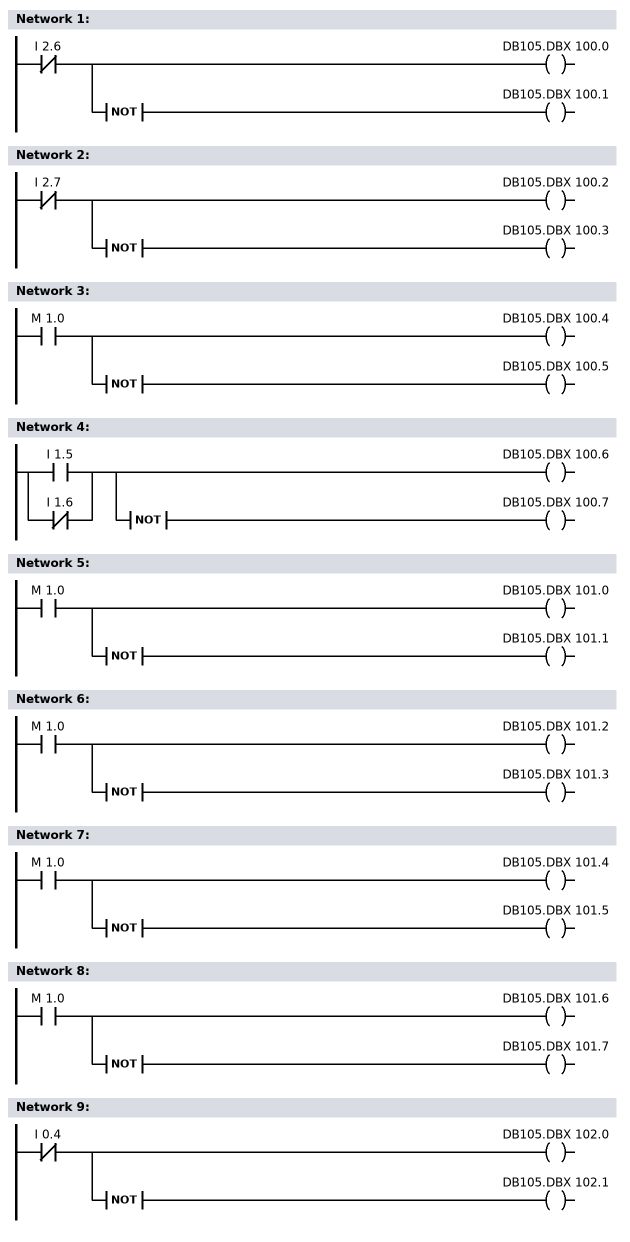
NETWORK
TITLE =
      AN    I 2.6;
      =     L 22.0;
      A     L 22.0;
      BLD   102;
      =     DB105.DBX 100.0;
      A     L 22.0;
      NOT;
      =     DB105.DBX 100.1;
NETWORK
TITLE =
      AN    I 2.7;
      =     L 22.0;
      A     L 22.0;
      BLD   102;
      =     DB105.DBX 100.2;
      A     L 22.0;
      NOT;
      =     DB105.DBX 100.3;
NETWORK
TITLE =
      A     M 1.0;
      =     L 22.0;
      A     L 22.0;
      BLD   102;
      =     DB105.DBX 100.4;
      A     L 22.0;
      NOT;
      =     DB105.DBX 100.5;
NETWORK
TITLE =
      O     I 1.5;
      ON    I 1.6;
      =     L 22.0;
      A     L 22.0;
      BLD   102;
      =     DB105.DBX 100.6;
      A     L 22.0;
      NOT;
      =     DB105.DBX 100.7;
NETWORK
TITLE =
      A     M 1.0;
      =     L 22.0;
      A     L 22.0;
      BLD   102;
      =     DB105.DBX 101.0;
      A     L 22.0;
      NOT;
      =     DB105.DBX 101.1;
NETWORK
TITLE =
      A     M 1.0;
      =     L 22.0;
      A     L 22.0;
      BLD   102;
      =     DB105.DBX 101.2;
      A     L 22.0;
      NOT;
      =     DB105.DBX 101.3;
NETWORK
TITLE =
      A     M 1.0;
      =     L 22.0;
      A     L 22.0;
      BLD   102;
      =     DB105.DBX 101.4;
      A     L 22.0;
      NOT;
      =     DB105.DBX 101.5;
NETWORK
TITLE =
      A     M 1.0;
      =     L 22.0;
      A     L 22.0;
      BLD   102;
      =     DB105.DBX 101.6;
      A     L 22.0;
      NOT;
      =     DB105.DBX 101.7;
NETWORK
TITLE =
      AN    I 0.4;
      =     L 22.0;
      A     L 22.0;
      BLD   102;
      =     DB105.DBX 102.0;
      A     L 22.0;
      NOT;
      =     DB105.DBX 102.1;
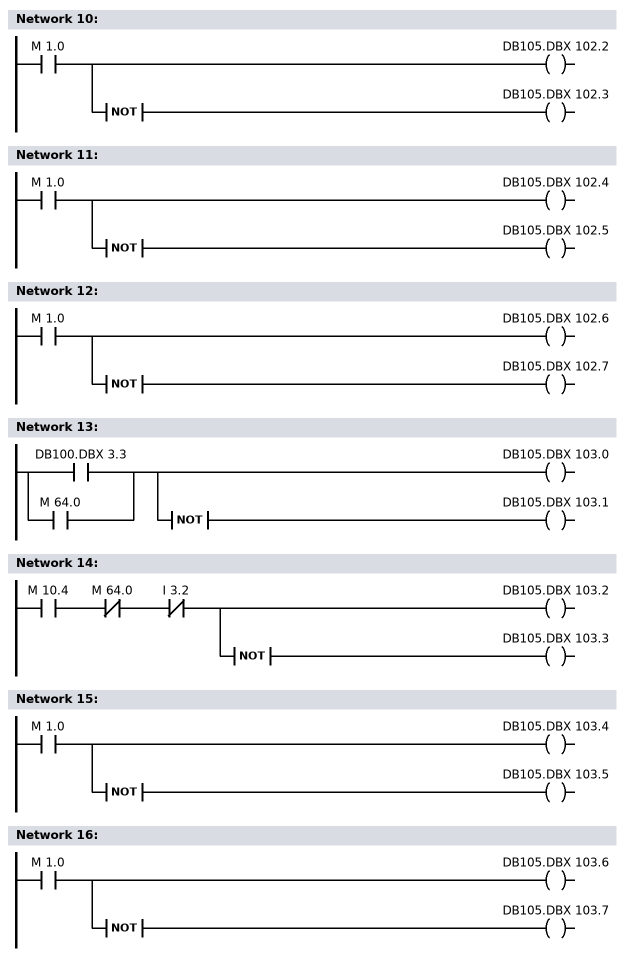
NETWORK
TITLE =
      A     M 1.0;
      =     L 22.0;
      A     L 22.0;
      BLD   102;
      =     DB105.DBX 102.2;
      A     L 22.0;
      NOT;
      =     DB105.DBX 102.3;
NETWORK
TITLE =
      A     M 1.0;
      =     L 22.0;
      A     L 22.0;
      BLD   102;
      =     DB105.DBX 102.4;
      A     L 22.0;
      NOT;
      =     DB105.DBX 102.5;
NETWORK
TITLE =
      A     M 1.0;
      =     L 22.0;
      A     L 22.0;
      BLD   102;
      =     DB105.DBX 102.6;
      A     L 22.0;
      NOT;
      =     DB105.DBX 102.7;
NETWORK
TITLE =
      O     DB100.DBX 3.3;
      O     M 64.0;
      =     L 22.0;
      A     L 22.0;
      BLD   102;
      =     DB105.DBX 103.0;
      A     L 22.0;
      NOT;
      =     DB105.DBX 103.1;
NETWORK
TITLE =
      A     M 10.4;
      AN    M 64.0;
      AN    I 3.2;
      =     L 22.0;
      A     L 22.0;
      BLD   102;
      =     DB105.DBX 103.2;
      A     L 22.0;
      NOT;
      =     DB105.DBX 103.3;
NETWORK
TITLE =
      A     M 1.0;
      =     L 22.0;
      A     L 22.0;
      BLD   102;
      =     DB105.DBX 103.4;
      A     L 22.0;
      NOT;
      =     DB105.DBX 103.5;
NETWORK
TITLE =
      A     M 1.0;
      =     L 22.0;
      A     L 22.0;
      BLD   102;
      =     DB105.DBX 103.6;
      A     L 22.0;
      NOT;
      =     DB105.DBX 103.7;
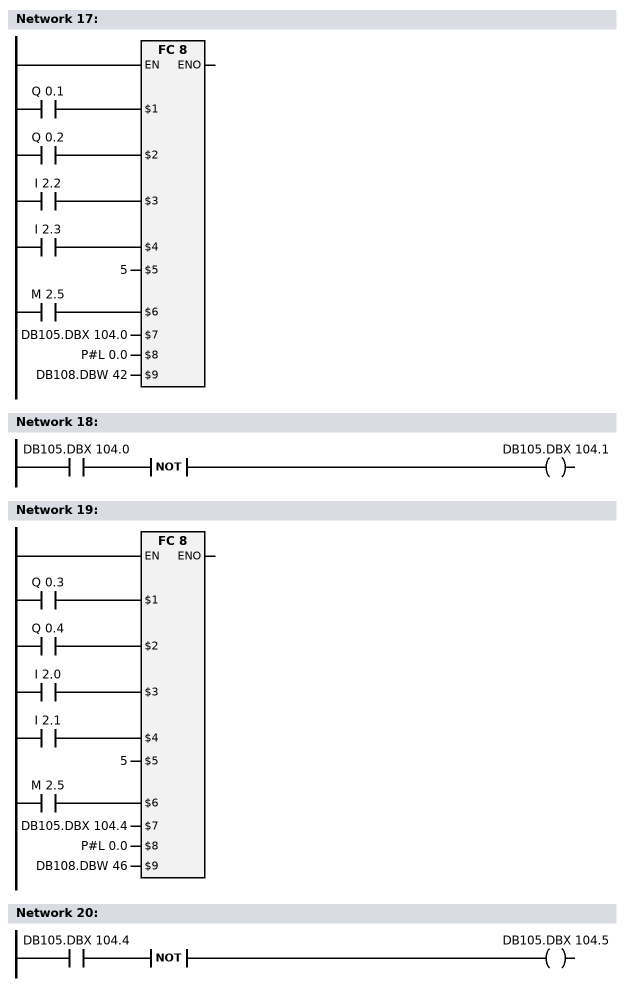
NETWORK
TITLE =
      A     Q 0.1;
      =     L 22.0;
      BLD   103;
      A     Q 0.2;
      =     L 22.1;
      BLD   103;
      A     I 2.2;
      =     L 22.2;
      BLD   103;
      A     I 2.3;
      =     L 22.3;
      BLD   103;
      A     M 2.5;
      =     L 22.4;
      BLD   103;
      CALL  FC 8 (
           $1                       := L 22.0,
           $2                       := L 22.1,
           $3                       := L 22.2,
           $4                       := L 22.3,
           $5                       := 5,
           $6                       := L 22.4,
           $7                       := DB105.DBX 104.0,
           $8                       := P#L 0.0,
           $9                       := DB108.DBW 42);
      NOP   0;
NETWORK
TITLE =
      A     DB105.DBX 104.0;
      NOT;
      =     DB105.DBX 104.1;
NETWORK
TITLE =
      A     Q 0.3;
      =     L 22.0;
      BLD   103;
      A     Q 0.4;
      =     L 22.1;
      BLD   103;
      A     I 2.0;
      =     L 22.2;
      BLD   103;
      A     I 2.1;
      =     L 22.3;
      BLD   103;
      A     M 2.5;
      =     L 22.4;
      BLD   103;
      CALL  FC 8 (
           $1                       := L 22.0,
           $2                       := L 22.1,
           $3                       := L 22.2,
           $4                       := L 22.3,
           $5                       := 5,
           $6                       := L 22.4,
           $7                       := DB105.DBX 104.4,
           $8                       := P#L 0.0,
           $9                       := DB108.DBW 46);
      NOP   0;
NETWORK
TITLE =
      A     DB105.DBX 104.4;
      NOT;
      =     DB105.DBX 104.5;
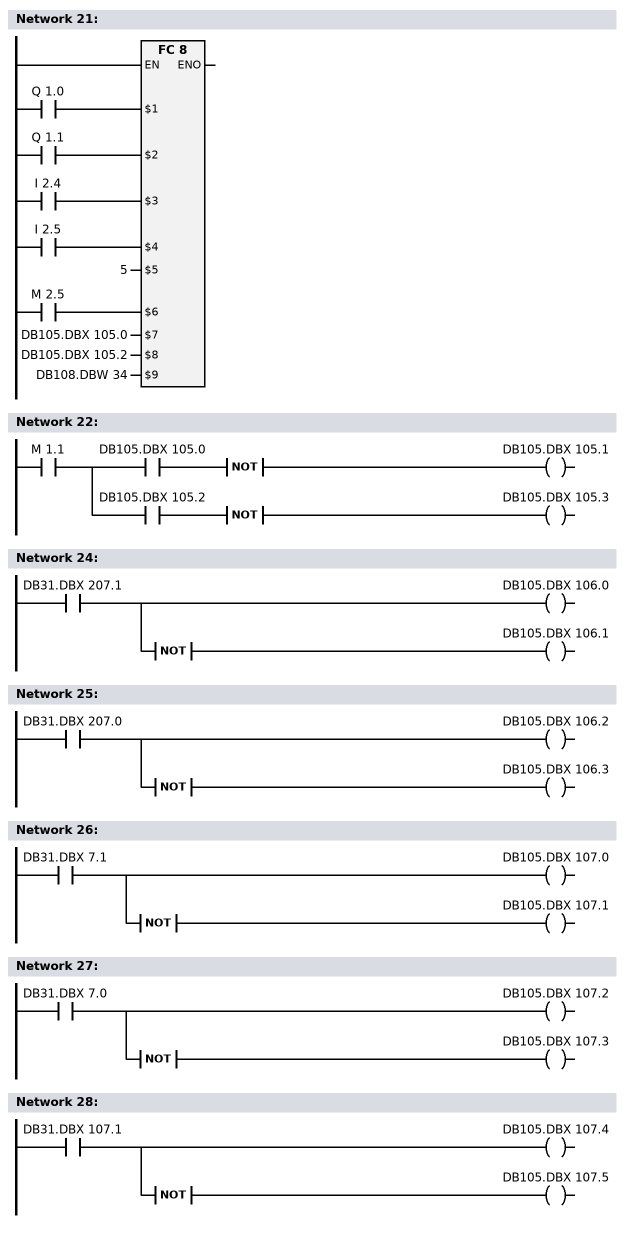
NETWORK
TITLE =
      A     Q 1.0;
      =     L 22.0;
      BLD   103;
      A     Q 1.1;
      =     L 22.1;
      BLD   103;
      A     I 2.4;
      =     L 22.2;
      BLD   103;
      A     I 2.5;
      =     L 22.3;
      BLD   103;
      A     M 2.5;
      =     L 22.4;
      BLD   103;
      CALL  FC 8 (
           $1                       := L 22.0,
           $2                       := L 22.1,
           $3                       := L 22.2,
           $4                       := L 22.3,
           $5                       := 5,
           $6                       := L 22.4,
           $7                       := DB105.DBX 105.0,
           $8                       := DB105.DBX 105.2,
           $9                       := DB108.DBW 34);
      NOP   0;
NETWORK
TITLE =
      A     M 1.1;
      =     L 22.0;
      A     L 22.0;
      A     DB105.DBX 105.0;
      NOT;
      =     DB105.DBX 105.1;
      A     L 22.0;
      A     DB105.DBX 105.2;
      NOT;
      =     DB105.DBX 105.3;
NETWORK
TITLE =
NETWORK
TITLE =
      A     DB31.DBX 207.1;
      =     L 22.0;
      A     L 22.0;
      BLD   102;
      =     DB105.DBX 106.0;
      A     L 22.0;
      NOT;
      =     DB105.DBX 106.1;
NETWORK
TITLE =
      A     DB31.DBX 207.0;
      =     L 22.0;
      A     L 22.0;
      BLD   102;
      =     DB105.DBX 106.2;
      A     L 22.0;
      NOT;
      =     DB105.DBX 106.3;
NETWORK
TITLE =
      A     DB31.DBX 7.1;
      =     L 22.0;
      A     L 22.0;
      BLD   102;
      =     DB105.DBX 107.0;
      A     L 22.0;
      NOT;
      =     DB105.DBX 107.1;
NETWORK
TITLE =
      A     DB31.DBX 7.0;
      =     L 22.0;
      A     L 22.0;
      BLD   102;
      =     DB105.DBX 107.2;
      A     L 22.0;
      NOT;
      =     DB105.DBX 107.3;
NETWORK
TITLE =
      A     DB31.DBX 107.1;
      =     L 22.0;
      A     L 22.0;
      BLD   102;
      =     DB105.DBX 107.4;
      A     L 22.0;
      NOT;
      =     DB105.DBX 107.5;
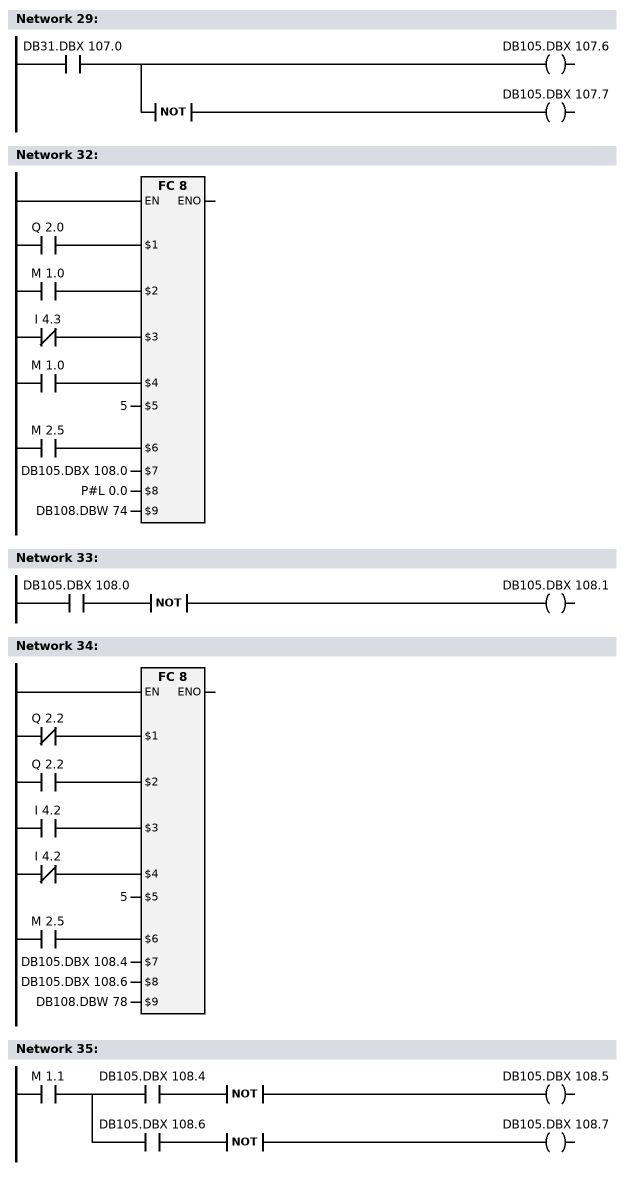
NETWORK
TITLE =
      A     DB31.DBX 107.0;
      =     L 22.0;
      A     L 22.0;
      BLD   102;
      =     DB105.DBX 107.6;
      A     L 22.0;
      NOT;
      =     DB105.DBX 107.7;
NETWORK
TITLE =
NETWORK
TITLE =
NETWORK
TITLE =
      A     Q 2.0;
      =     L 22.0;
      BLD   103;
      A     M 1.0;
      =     L 22.1;
      BLD   103;
      AN    I 4.3;
      =     L 22.2;
      BLD   103;
      A     M 1.0;
      =     L 22.3;
      BLD   103;
      A     M 2.5;
      =     L 22.4;
      BLD   103;
      CALL  FC 8 (
           $1                       := L 22.0,
           $2                       := L 22.1,
           $3                       := L 22.2,
           $4                       := L 22.3,
           $5                       := 5,
           $6                       := L 22.4,
           $7                       := DB105.DBX 108.0,
           $8                       := P#L 0.0,
           $9                       := DB108.DBW 74);
      NOP   0;
NETWORK
TITLE =
      A     DB105.DBX 108.0;
      NOT;
      =     DB105.DBX 108.1;
NETWORK
TITLE =
      AN    Q 2.2;
      =     L 22.0;
      BLD   103;
      A     Q 2.2;
      =     L 22.1;
      BLD   103;
      A     I 4.2;
      =     L 22.2;
      BLD   103;
      AN    I 4.2;
      =     L 22.3;
      BLD   103;
      A     M 2.5;
      =     L 22.4;
      BLD   103;
      CALL  FC 8 (
           $1                       := L 22.0,
           $2                       := L 22.1,
           $3                       := L 22.2,
           $4                       := L 22.3,
           $5                       := 5,
           $6                       := L 22.4,
           $7                       := DB105.DBX 108.4,
           $8                       := DB105.DBX 108.6,
           $9                       := DB108.DBW 78);
      NOP   0;
NETWORK
TITLE =
      A     M 1.1;
      =     L 22.0;
      A     L 22.0;
      A     DB105.DBX 108.4;
      NOT;
      =     DB105.DBX 108.5;
      A     L 22.0;
      A     DB105.DBX 108.6;
      NOT;
      =     DB105.DBX 108.7;
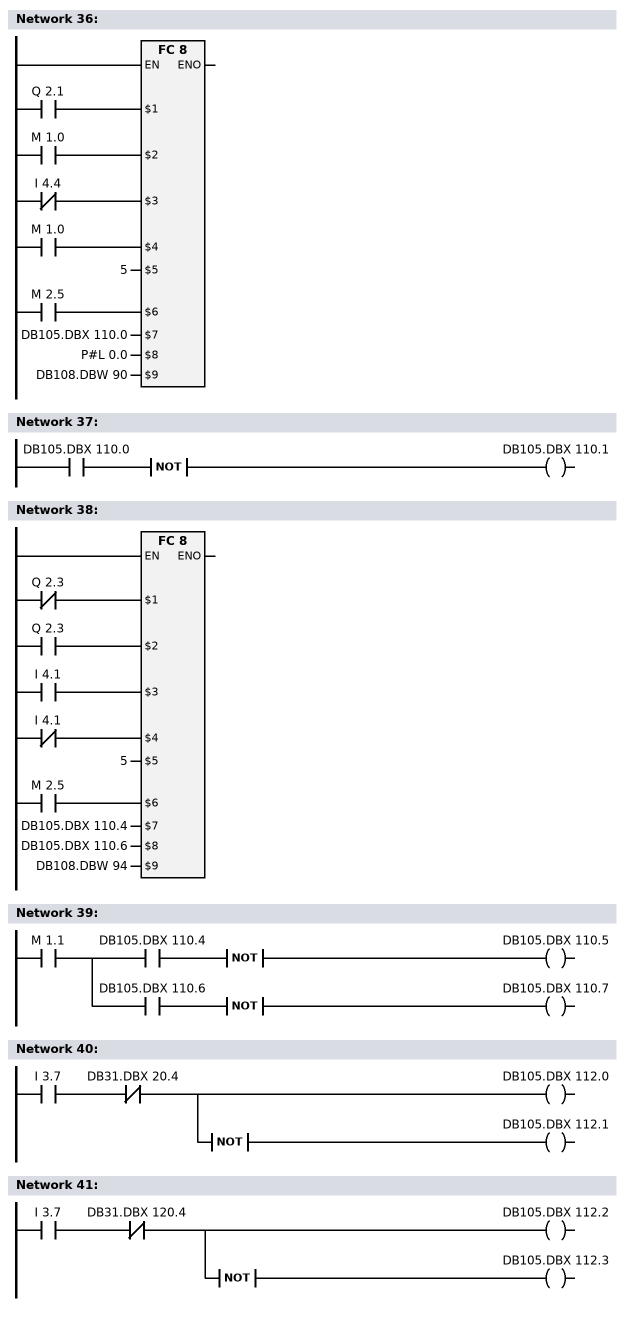
NETWORK
TITLE =
      A     Q 2.1;
      =     L 22.0;
      BLD   103;
      A     M 1.0;
      =     L 22.1;
      BLD   103;
      AN    I 4.4;
      =     L 22.2;
      BLD   103;
      A     M 1.0;
      =     L 22.3;
      BLD   103;
      A     M 2.5;
      =     L 22.4;
      BLD   103;
      CALL  FC 8 (
           $1                       := L 22.0,
           $2                       := L 22.1,
           $3                       := L 22.2,
           $4                       := L 22.3,
           $5                       := 5,
           $6                       := L 22.4,
           $7                       := DB105.DBX 110.0,
           $8                       := P#L 0.0,
           $9                       := DB108.DBW 90);
      NOP   0;
NETWORK
TITLE =
      A     DB105.DBX 110.0;
      NOT;
      =     DB105.DBX 110.1;
NETWORK
TITLE =
      AN    Q 2.3;
      =     L 22.0;
      BLD   103;
      A     Q 2.3;
      =     L 22.1;
      BLD   103;
      A     I 4.1;
      =     L 22.2;
      BLD   103;
      AN    I 4.1;
      =     L 22.3;
      BLD   103;
      A     M 2.5;
      =     L 22.4;
      BLD   103;
      CALL  FC 8 (
           $1                       := L 22.0,
           $2                       := L 22.1,
           $3                       := L 22.2,
           $4                       := L 22.3,
           $5                       := 5,
           $6                       := L 22.4,
           $7                       := DB105.DBX 110.4,
           $8                       := DB105.DBX 110.6,
           $9                       := DB108.DBW 94);
      NOP   0;
NETWORK
TITLE =
      A     M 1.1;
      =     L 22.0;
      A     L 22.0;
      A     DB105.DBX 110.4;
      NOT;
      =     DB105.DBX 110.5;
      A     L 22.0;
      A     DB105.DBX 110.6;
      NOT;
      =     DB105.DBX 110.7;
NETWORK
TITLE =
      A     I 3.7;
      AN    DB31.DBX 20.4;
      =     L 22.0;
      A     L 22.0;
      BLD   102;
      =     DB105.DBX 112.0;
      A     L 22.0;
      NOT;
      =     DB105.DBX 112.1;
NETWORK
TITLE =
      A     I 3.7;
      AN    DB31.DBX 120.4;
      =     L 22.0;
      A     L 22.0;
      BLD   102;
      =     DB105.DBX 112.2;
      A     L 22.0;
      NOT;
      =     DB105.DBX 112.3;
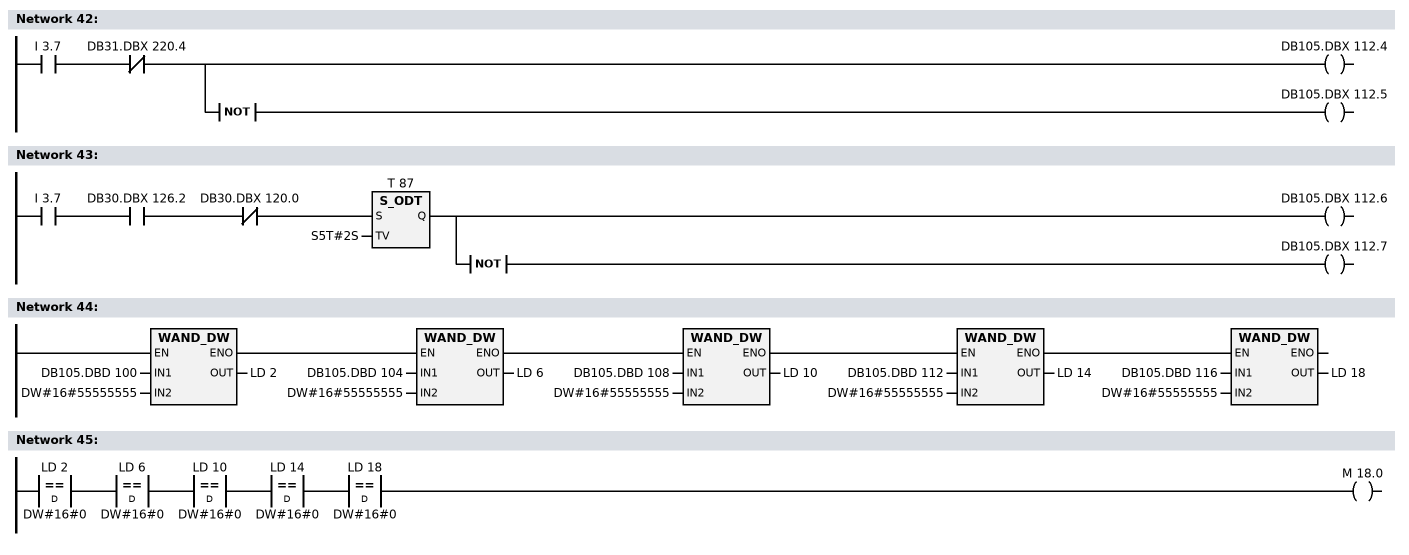
NETWORK
TITLE =
      A     I 3.7;
      AN    DB31.DBX 220.4;
      =     L 22.0;
      A     L 22.0;
      BLD   102;
      =     DB105.DBX 112.4;
      A     L 22.0;
      NOT;
      =     DB105.DBX 112.5;
NETWORK
TITLE =
      A     I 3.7;
      A     DB30.DBX 126.2;
      AN    DB30.DBX 120.0;
      L     S5T#2S;
      SD    T 87;
      NOP   0;
      NOP   0;
      NOP   0;
      A     T 87;
      =     L 22.0;
      A     L 22.0;
      BLD   102;
      =     DB105.DBX 112.6;
      A     L 22.0;
      NOT;
      =     DB105.DBX 112.7;
NETWORK
TITLE =
      A(;
      A(;
      A(;
      A(;
      L     DB105.DBD 100;
      L     DW#16#55555555;
      AD;
      T     LD 2;
      SET;
      SAVE;
      CLR;
      A     BR;
      );
      JNB   M001;
      L     DB105.DBD 104;
      L     DW#16#55555555;
      AD;
      T     LD 6;
      SET;
      SAVE;
      CLR;
M001: A     BR;
      );
      JNB   M002;
      L     DB105.DBD 108;
      L     DW#16#55555555;
      AD;
      T     LD 10;
      SET;
      SAVE;
      CLR;
M002: A     BR;
      );
      JNB   M003;
      L     DB105.DBD 112;
      L     DW#16#55555555;
      AD;
      T     LD 14;
      SET;
      SAVE;
      CLR;
M003: A     BR;
      );
      JNB   M004;
      L     DB105.DBD 116;
      L     DW#16#55555555;
      AD;
      T     LD 18;
M004: NOP   0;
NETWORK
TITLE =
      A(;
      L     LD 2;
      L     DW#16#0;
      ==D;
      );
      A(;
      L     LD 6;
      L     DW#16#0;
      ==D;
      );
      A(;
      L     LD 10;
      L     DW#16#0;
      ==D;
      );
      A(;
      L     LD 14;
      L     DW#16#0;
      ==D;
      );
      A(;
      L     LD 18;
      L     DW#16#0;
      ==D;
      );
      =     M 18.0;
END_FUNCTION

FUNCTION FC 119 : VOID
VERSION : 0.1
BEGIN
// (block stored without names or comments; labels and parameter names are numbered)
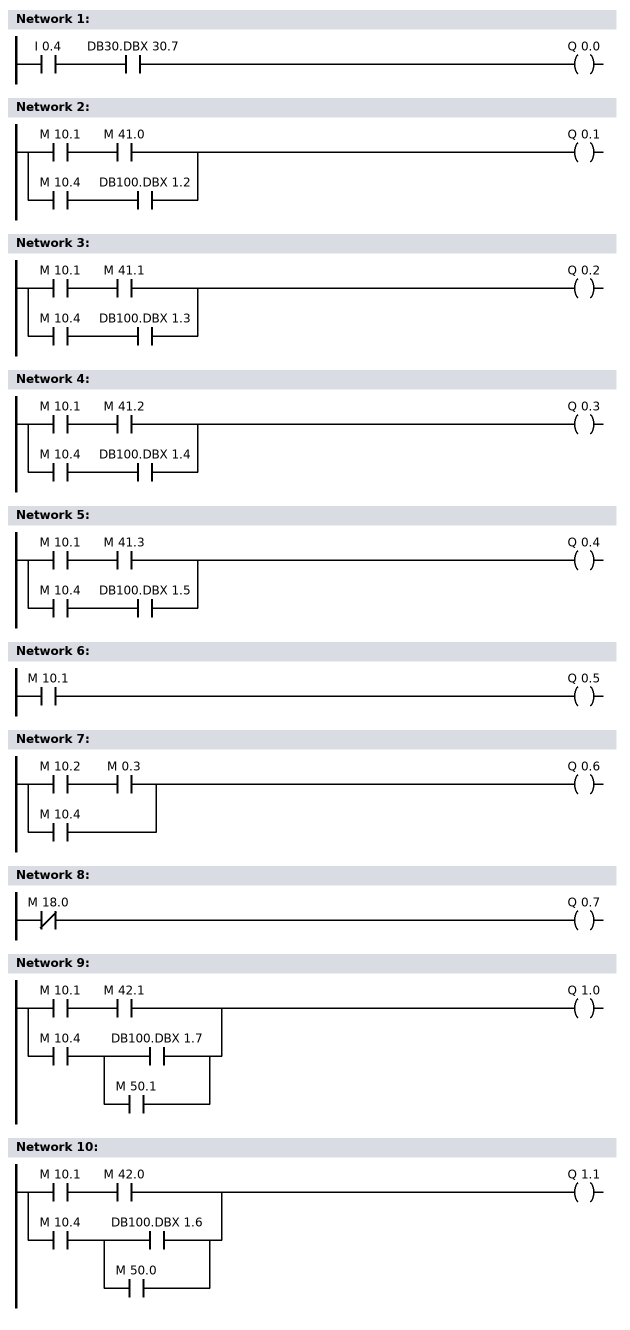
NETWORK
TITLE =
      A     I 0.4;
      A     DB30.DBX 30.7;
      =     Q 0.0;
NETWORK
TITLE =
      A     M 10.1;
      A     M 41.0;
      O;
      A     M 10.4;
      A     DB100.DBX 1.2;
      =     Q 0.1;
NETWORK
TITLE =
      A     M 10.1;
      A     M 41.1;
      O;
      A     M 10.4;
      A     DB100.DBX 1.3;
      =     Q 0.2;
NETWORK
TITLE =
      A     M 10.1;
      A     M 41.2;
      O;
      A     M 10.4;
      A     DB100.DBX 1.4;
      =     Q 0.3;
NETWORK
TITLE =
      A     M 10.1;
      A     M 41.3;
      O;
      A     M 10.4;
      A     DB100.DBX 1.5;
      =     Q 0.4;
NETWORK
TITLE =
      A     M 10.1;
      =     Q 0.5;
NETWORK
TITLE =
      A     M 10.2;
      A     M 0.3;
      O     M 10.4;
      =     Q 0.6;
NETWORK
TITLE =
      AN    M 18.0;
      =     Q 0.7;
NETWORK
TITLE =
      A     M 10.1;
      A     M 42.1;
      O;
      A     M 10.4;
      A(;
      O     DB100.DBX 1.7;
      O     M 50.1;
      );
      =     Q 1.0;
NETWORK
TITLE =
      A     M 10.1;
      A     M 42.0;
      O;
      A     M 10.4;
      A(;
      O     DB100.DBX 1.6;
      O     M 50.0;
      );
      =     Q 1.1;
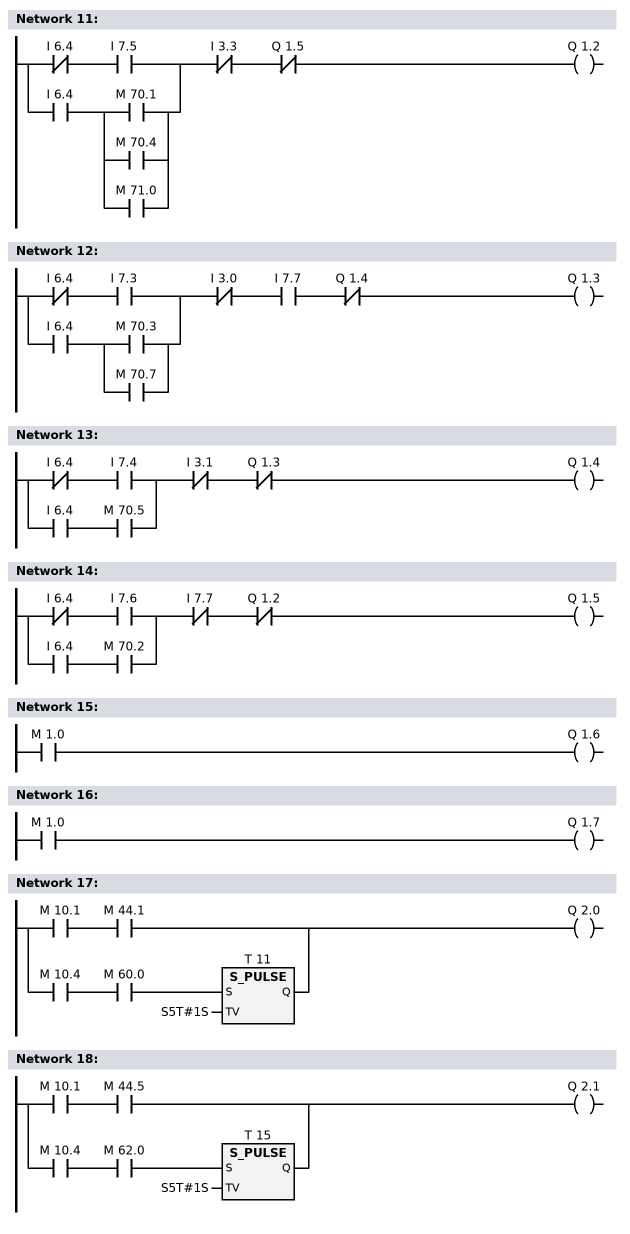
NETWORK
TITLE =
      A(;
      AN    I 6.4;
      A     I 7.5;
      O;
      A     I 6.4;
      A(;
      O     M 70.1;
      O     M 70.4;
      O     M 71.0;
      );
      );
      AN    I 3.3;
      AN    Q 1.5;
      =     Q 1.2;
NETWORK
TITLE =
      A(;
      AN    I 6.4;
      A     I 7.3;
      O;
      A     I 6.4;
      A(;
      O     M 70.3;
      O     M 70.7;
      );
      );
      AN    I 3.0;
      A     I 7.7;
      AN    Q 1.4;
      =     Q 1.3;
NETWORK
TITLE =
      A(;
      AN    I 6.4;
      A     I 7.4;
      O;
      A     I 6.4;
      A     M 70.5;
      );
      AN    I 3.1;
      AN    Q 1.3;
      =     Q 1.4;
NETWORK
TITLE =
      A(;
      AN    I 6.4;
      A     I 7.6;
      O;
      A     I 6.4;
      A     M 70.2;
      );
      AN    I 7.7;
      AN    Q 1.2;
      =     Q 1.5;
NETWORK
TITLE =
      A     M 1.0;
      =     Q 1.6;
NETWORK
TITLE =
      A     M 1.0;
      =     Q 1.7;
NETWORK
TITLE =
      A     M 10.1;
      A     M 44.1;
      O(;
      A     M 10.4;
      A     M 60.0;
      L     S5T#1S;
      SP    T 11;
      NOP   0;
      NOP   0;
      NOP   0;
      A     T 11;
      );
      =     Q 2.0;
NETWORK
TITLE =
      A     M 10.1;
      A     M 44.5;
      O(;
      A     M 10.4;
      A     M 62.0;
      L     S5T#1S;
      SP    T 15;
      NOP   0;
      NOP   0;
      NOP   0;
      A     T 15;
      );
      =     Q 2.1;
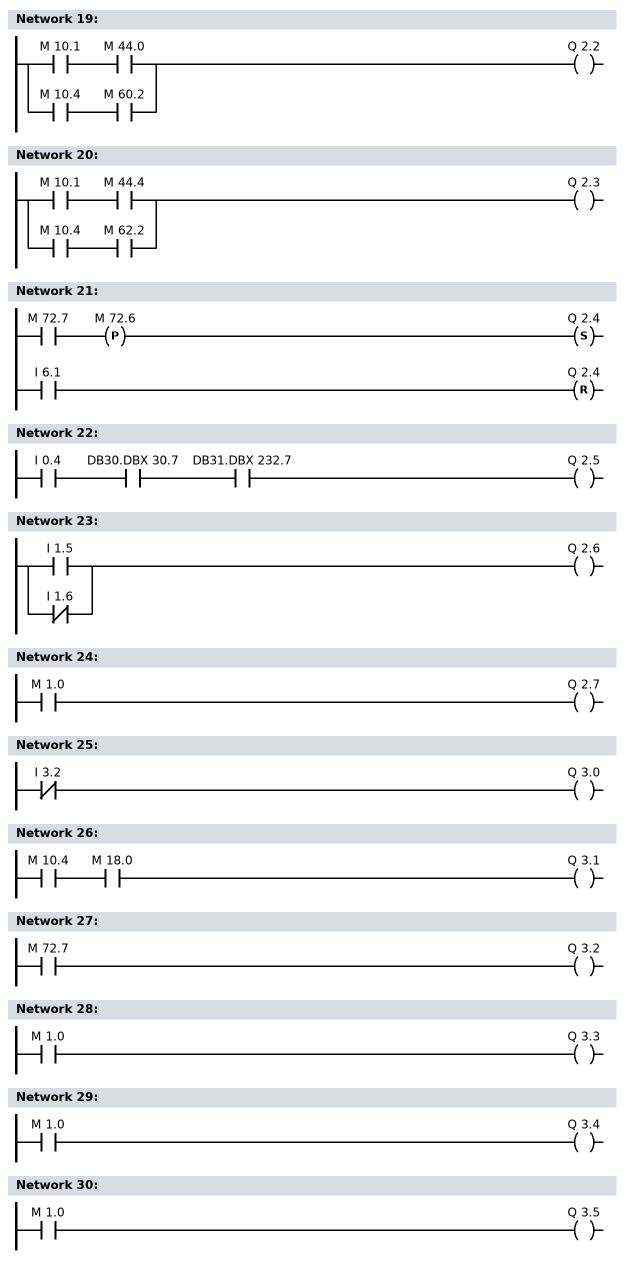
NETWORK
TITLE =
      A     M 10.1;
      A     M 44.0;
      O;
      A     M 10.4;
      A     M 60.2;
      =     Q 2.2;
NETWORK
TITLE =
      A     M 10.1;
      A     M 44.4;
      O;
      A     M 10.4;
      A     M 62.2;
      =     Q 2.3;
NETWORK
TITLE =
      A     M 72.7;
      FP    M 72.6;
      S     Q 2.4;
      A     I 6.1;
      R     Q 2.4;
      NOP   0;
NETWORK
TITLE =
      A     I 0.4;
      A     DB30.DBX 30.7;
      A     DB31.DBX 232.7;
      =     Q 2.5;
NETWORK
TITLE =
      O     I 1.5;
      ON    I 1.6;
      =     Q 2.6;
NETWORK
TITLE =
      A     M 1.0;
      =     Q 2.7;
NETWORK
TITLE =
      AN    I 3.2;
      =     Q 3.0;
NETWORK
TITLE =
      A     M 10.4;
      A     M 18.0;
      =     Q 3.1;
NETWORK
TITLE =
      A     M 72.7;
      =     Q 3.2;
NETWORK
TITLE =
      A     M 1.0;
      =     Q 3.3;
NETWORK
TITLE =
      A     M 1.0;
      =     Q 3.4;
NETWORK
TITLE =
      A     M 1.0;
      =     Q 3.5;
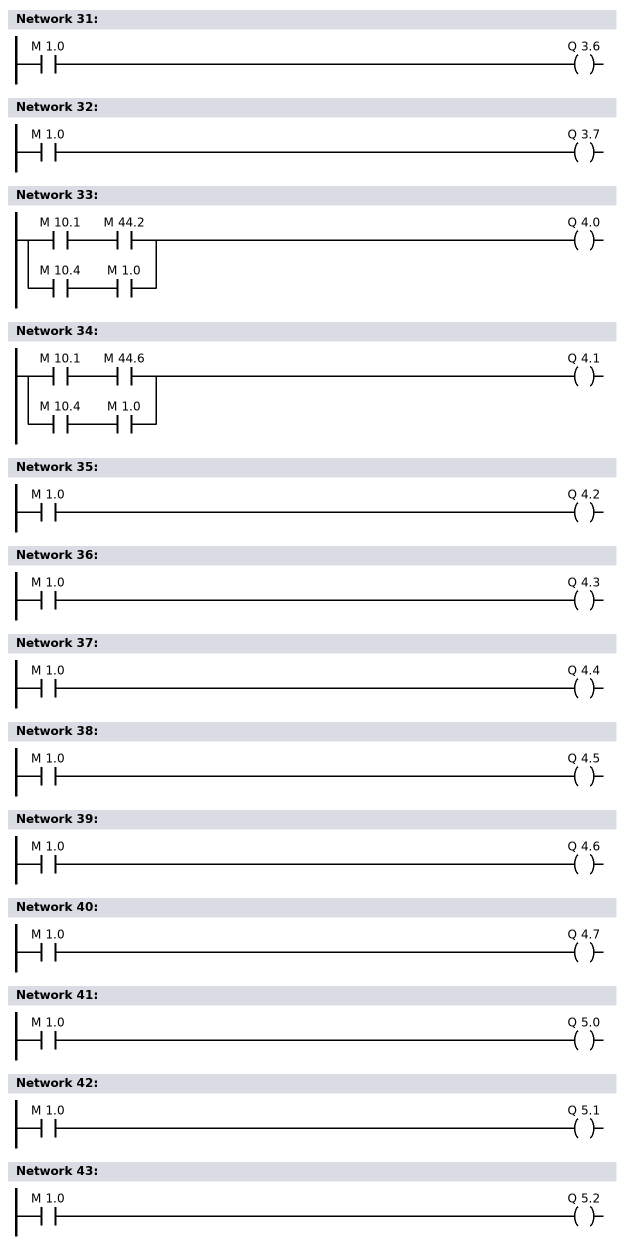
NETWORK
TITLE =
      A     M 1.0;
      =     Q 3.6;
NETWORK
TITLE =
      A     M 1.0;
      =     Q 3.7;
NETWORK
TITLE =
      A     M 10.1;
      A     M 44.2;
      O;
      A     M 10.4;
      A     M 1.0;
      =     Q 4.0;
NETWORK
TITLE =
      A     M 10.1;
      A     M 44.6;
      O;
      A     M 10.4;
      A     M 1.0;
      =     Q 4.1;
NETWORK
TITLE =
      A     M 1.0;
      =     Q 4.2;
NETWORK
TITLE =
      A     M 1.0;
      =     Q 4.3;
NETWORK
TITLE =
      A     M 1.0;
      =     Q 4.4;
NETWORK
TITLE =
      A     M 1.0;
      =     Q 4.5;
NETWORK
TITLE =
      A     M 1.0;
      =     Q 4.6;
NETWORK
TITLE =
      A     M 1.0;
      =     Q 4.7;
NETWORK
TITLE =
      A     M 1.0;
      =     Q 5.0;
NETWORK
TITLE =
      A     M 1.0;
      =     Q 5.1;
NETWORK
TITLE =
      A     M 1.0;
      =     Q 5.2;
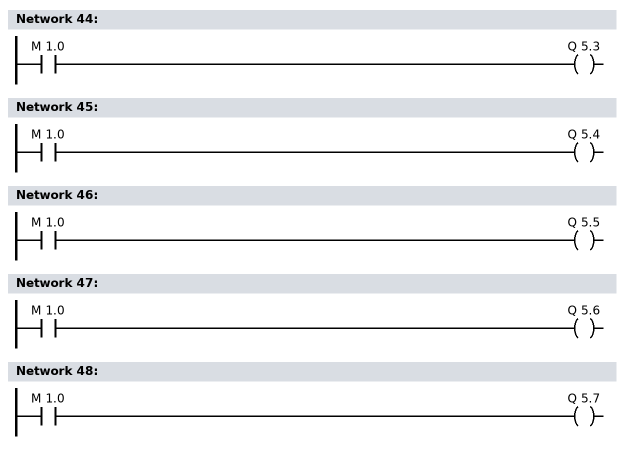
NETWORK
TITLE =
      A     M 1.0;
      =     Q 5.3;
NETWORK
TITLE =
      A     M 1.0;
      =     Q 5.4;
NETWORK
TITLE =
      A     M 1.0;
      =     Q 5.5;
NETWORK
TITLE =
      A     M 1.0;
      =     Q 5.6;
NETWORK
TITLE =
      A     M 1.0;
      =     Q 5.7;
END_FUNCTION

DATA_BLOCK DB 2
VERSION : 0.0
BEGIN
// 66 bytes; values not shown
END_DATA_BLOCK

// DB 7: know-how protected block, not included

DATA_BLOCK DB 15
AUTHOR : AuD_MCE8
FAMILY : FM357_2
NAME : BF_DB15
VERSION : 2.1
FB 6
BEGIN
END_DATA_BLOCK

// DB 16: know-how protected block, not included

// DB 17: know-how protected block, not included

// DB 19: know-how protected block, not included

// DB 20: know-how protected block, not included

DATA_BLOCK DB 30
VERSION : 0.1
BEGIN
// 962 bytes; values not shown
END_DATA_BLOCK

DATA_BLOCK DB 31
VERSION : 0.1
BEGIN
// 500 bytes; values not shown
END_DATA_BLOCK

DATA_BLOCK DB 100
VERSION : 0.1
BEGIN
// 14 bytes; values not shown
END_DATA_BLOCK

DATA_BLOCK DB 105
VERSION : 0.0
BEGIN
// 148 bytes; values not shown
END_DATA_BLOCK

DATA_BLOCK DB 108
VERSION : 0.1
BEGIN
// 402 bytes; values not shown
END_DATA_BLOCK

DATA_BLOCK DB 110
VERSION : 0.1
BEGIN
// 4206 bytes; values not shown
END_DATA_BLOCK

DATA_BLOCK DB 115
AUTHOR : AuD_MCE8
FAMILY : FM357_2
NAME : USERDB
VERSION : 3.1
BEGIN
// 94 bytes; values not shown
END_DATA_BLOCK

DATA_BLOCK DB 121
AUTHOR : AuD_MCE8
FAMILY : FM357_2
NAME : VAR_ADDR
VERSION : 3.1
BEGIN
// 190 bytes; values not shown
END_DATA_BLOCK

DATA_BLOCK DB 141
AUTHOR : AuD_MCE8
FAMILY : FM357_2
VERSION : 0.0
FB 3
BEGIN
END_DATA_BLOCK

DATA_BLOCK DB 142
AUTHOR : AuD_MCE8
FAMILY : FM357_2
VERSION : 0.0
FB 3
BEGIN
END_DATA_BLOCK

DATA_BLOCK DB 143
AUTHOR : AuD_MCE8
FAMILY : FM357_2
VERSION : 0.0
FB 3
BEGIN
END_DATA_BLOCK

ORGANIZATION_BLOCK OB 1
VERSION : 1.0
BEGIN
// (block stored without names or comments; labels and parameter names are numbered)
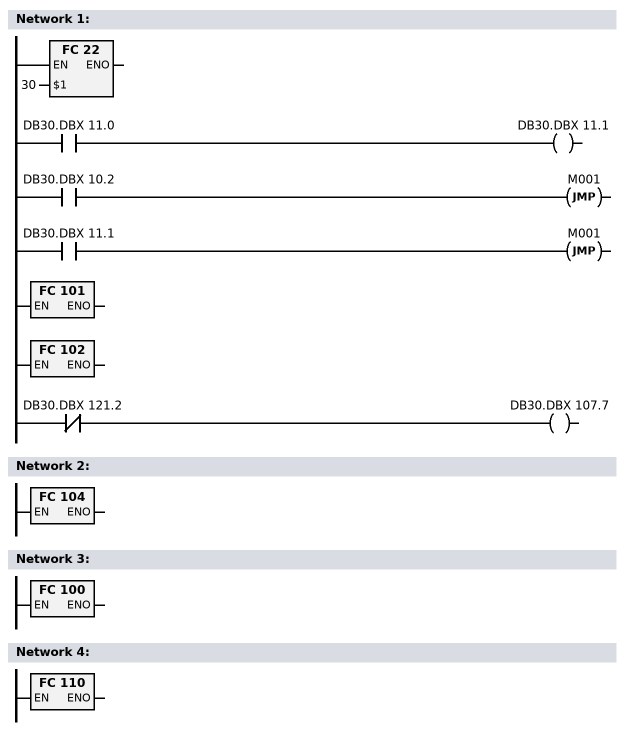
NETWORK
TITLE =
      CALL  FC 22 (
           $1                       := 30);
      A     DB30.DBX 11.0;
      =     DB30.DBX 11.1;
      A     DB30.DBX 10.2;
      JC    M001;
      A     DB30.DBX 11.1;
      JC    M001;
      CALL  FC 101;
      CALL  FC 102;
M001: NOP   0;
      AN    DB30.DBX 121.2;
      =     DB30.DBX 107.7;
      NOP   0;
NETWORK
TITLE =
      CALL  FC 104;
      NOP   0;
NETWORK
TITLE =
      CALL  FC 100;
      NOP   0;
NETWORK
TITLE =
      CALL  FC 110;
      NOP   0;
END_ORGANIZATION_BLOCK

ORGANIZATION_BLOCK OB 82
VERSION : 1.0
BEGIN
// (block stored without names or comments; labels and parameter names are numbered)
NETWORK
TITLE =
      CALL  FC 5 (
           $1                       := 30);
      BE;
END_ORGANIZATION_BLOCK

ORGANIZATION_BLOCK OB 100
VERSION : 1.0
BEGIN
// (block stored without names or comments; labels and parameter names are numbered)
NETWORK
TITLE =
      CALL  FC 1 (
           $1                       := 30,
           $2                       := 300,
           $3                       := 100,
           $4                       := TRUE,
           $5                       := TRUE);
      BE;
END_ORGANIZATION_BLOCK
